FUNCTION_BLOCK Tank1_1
VAR_INPUT
	//bSwitchFill : BOOL;
	bSwitchSink : BOOL;
END_VAR
VAR_IN_OUT
	bSwitchFill : BOOL;
END_VAR
VAR_OUTPUT
END_VAR
VAR
	bShl : BOOL := FALSE;
	bSll : BOOL := TRUE;
	nState : INT;
	level: INT := 3;
	tTime : TON;
	rTrig : R_TRIG;	
	
END_VAR



CASE nState OF
	
	0:	
		IF  NOT bSwitchSink THEN
			IF bSll THEN
				bSwitchFill := TRUE;
			END_IF
			(*IF NOT bShl THEN
				bSwitchFill := TRUE;
			END_IF*)
			tTime(IN := bSwitchFill,PT := T#1S);
			rTrig(CLK := tTime.Q);
			IF rTrig.Q THEN
				level := level + 2;
				tTime(IN := FALSE);
				IF level >= 5 THEN
					bSll := FALSE;
				END_IF
				IF level = 100 THEN
					bShl := TRUE;
					bSwitchFill := FALSE;
					nState := 10;
				END_IF
			END_IF
		 		
		ELSE
			IF NOT bSwitchFill THEN
				nState := 10;
			ELSE
				IF bSll THEN
					bSwitchFill := TRUE;
				END_IF
				(*IF NOT bShl THEN
					bSwitchFill := TRUE;
				END_IF*)
				tTime(IN := bSwitchFill,PT := T#1S);
				rTrig(CLK := tTime.Q);
				IF rTrig.Q THEN
					level := level + 1;
					tTime(IN := FALSE);
					IF level >= 5 THEN
						bSll := FALSE;
					END_IF
					IF level = 100 THEN
						bShl := TRUE;
						bSwitchFill := FALSE;
						nState := 10;
					END_IF
				END_IF
			END_IF
		END_IF
		
	10: 
		
		IF  bSwitchSink THEN
			IF bShl THEN
				bSwitchFill := FALSE;
			END_IF
			IF level > 90 THEN
				bSwitchFill := FALSE;
			ELSIF level <= 90 THEN
				bSwitchFill := bSwitchFill;
			END_IF
			IF NOT bSwitchFill THEN
				tTime(IN := bSwitchSink,PT := T#1S);
				rTrig(CLK := tTime.Q);
				IF rTrig.q THEN
					tTime(IN := FALSE);
					level := level - 1;
					IF level <> 100 THEN
						bShl := FALSE;
					END_IF
					IF level < 5 THEN
						bSwitchSink := FALSE;
						bSll := TRUE;
						nState := 0;
					END_IF
				END_IF
			ELSE
				IF level <> 100 THEN
					bShl := FALSE;
				END_IF
				nState := 0;
			END_IF
		ELSE
			IF NOT bSwitchFill THEN
				nState := 10;
			ELSE
				nState := 0;
			END_IF		
		END_IF
					
END_CASE

END_FUNCTION_BLOCK

(* stored: Version 1.1.0.1, ProductVersion 3.1.4024.0
   POU Tank1_1: Id {7d9ec4ef-88e1-453f-b1b5-ca44d24471b8}, SpecialFunc None *)
